// Mitsubishi GX Works2 project: 1   PLC: FX3G

PROGRAM MAIN
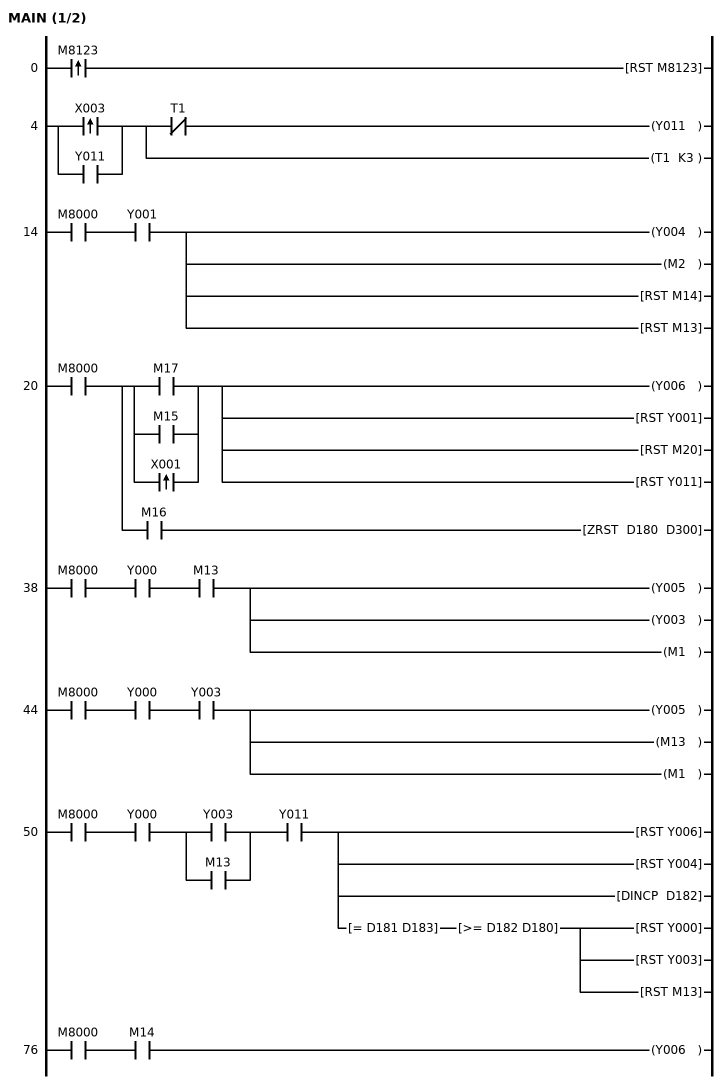
0     LDP     M8123
      RST     M8123
4     LDP     X003
      OR      Y011
      MPS
      ANI     T1
      OUT     Y011
      MPP
      OUT     T1 K3
14    LD      M8000
      AND     Y001
      OUT     Y004
      OUT     M2
      RST     M14
      RST     M13
20    LD      M8000
      MPS
      LD      M17
      OR      M15
      ORP     X001
      ANB
      OUT     Y006
      RST     Y001
      RST     M20
      RST     Y011
      MPP
      AND     M16
      ZRST    D180 D300
38    LD      M8000
      AND     Y000
      AND     M13
      OUT     Y005
      OUT     Y003
      OUT     M1
44    LD      M8000
      AND     Y000
      AND     Y003
      OUT     Y005
      OUT     M13
      OUT     M1
50    LD      M8000
      AND     Y000
      LD      Y003
      OR      M13
      ANB
      AND     Y011
      RST     Y006
      RST     Y004
      DINCP   D182
      AND=    D181 D183
      AND>=   D182 D180
      RST     Y000
      RST     Y003
      RST     M13
76    LD      M8000
      AND     M14
      OUT     Y006
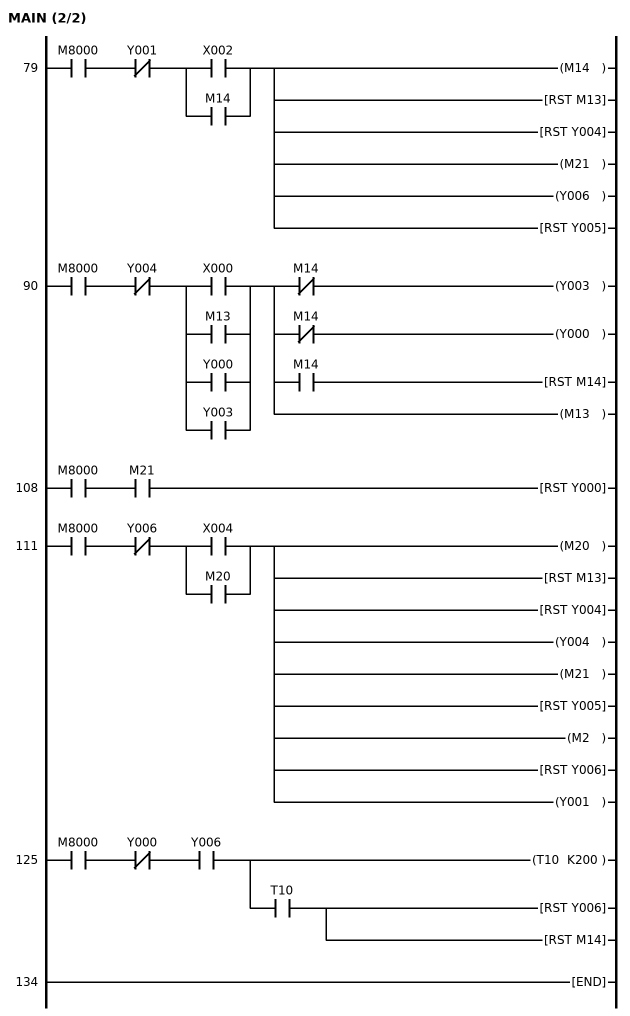
79    LD      M8000
      ANI     Y001
      LD      X002
      OR      M14
      ANB
      OUT     M14
      RST     M13
      RST     Y004
      OUT     M21
      OUT     Y006
      RST     Y005
90    LD      M8000
      ANI     Y004
      LD      X000
      OR      M13
      OR      Y000
      OR      Y003
      ANB
      MPS
      ANI     M14
      OUT     Y003
      MRD
      ANI     M14
      OUT     Y000
      MRD
      AND     M14
      RST     M14
      MPP
      OUT     M13
108   LD      M8000
      AND     M21
      RST     Y000
111   LD      M8000
      ANI     Y006
      LD      X004
      OR      M20
      ANB
      OUT     M20
      RST     M13
      RST     Y004
      OUT     Y004
      OUT     M21
      RST     Y005
      OUT     M2
      RST     Y006
      OUT     Y001
125   LD      M8000
      ANI     Y000
      AND     Y006
      OUT     T10 K200
      AND     T10
      RST     Y006
      RST     M14
134   END
END_PROGRAM
